PROGRAM S3_01_Motion_43
VAR
	HMI_Motion: FB_HMI_Control;
	Motion: FB_Motion2way;

	tMessageOffset: UINT;
	tNumMessagesPerRow: UINT;
	
	
	MyAdvanceInterlock: BOOL;
	MyReturnInterlock: BOOL;
	
	MyAutoAdvanceCondition: BOOL;
	MyAutoReturnCondition: BOOL;
	testword: WORD;
	myAdvancePrompt: BOOL;
	myReturnPrompt: BOOL;
	advancedSensor: BOOL;
	returnedSensor: BOOL;
	AdvanceCoil: BOOL;
	ReturnCoil: BOOL;
END_VAR

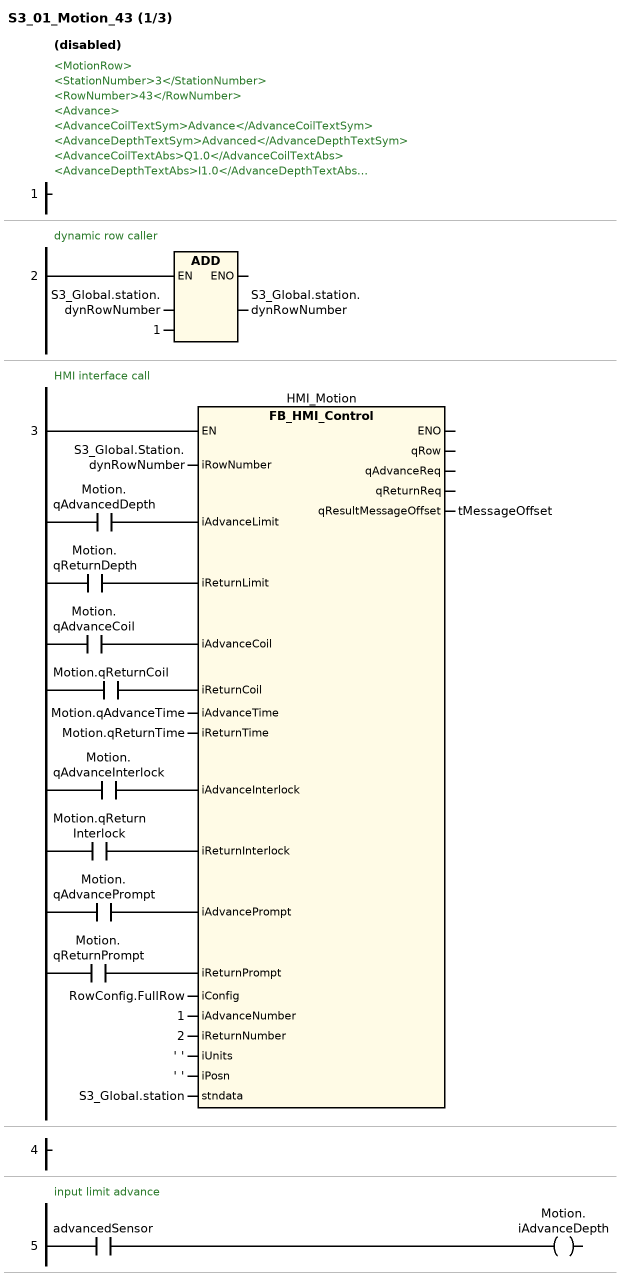
// NETWORK 1 (disabled)
// <MotionRow>
// <StationNumber>3</StationNumber>
// <RowNumber>43</RowNumber>
//   <Advance>
//     <AdvanceCoilTextSym>Advance</AdvanceCoilTextSym>
//     <AdvanceDepthTextSym>Advanced</AdvanceDepthTextSym>
//     <AdvanceCoilTextAbs>Q1.0</AdvanceCoilTextAbs>
//     <AdvanceDepthTextAbs>I1.0</AdvanceDepthTextAbs>
//     <ManSeq>1</ManSeq>
//   </Advance>
//   <Return>
//     <ReturnCoilTextSym>Return</ReturnCoilTextSym>
//     <ReturnDepthTextSym>Returned</ReturnDepthTextSym>
//     <ReturnCoilTextAbs>Q1.1</ReturnCoilTextAbs>
//     <ReturnDepthTextAbs>I1.1</ReturnDepthTextAbs>
//    <ManSeq>2</ManSeq>
//   </Return>
//   <Motion>
//     <NameSym>Clamp Cylinder</NameSym>
//     <NameAbs>A1</NameAbs>
//   </Motion>
// </MotionRow>

// NETWORK 2
// dynamic row caller
S3_Global.station.dynRowNumber := S3_Global.station.dynRowNumber + 1;

// NETWORK 3
// HMI interface call
HMI_Motion(
    iRowNumber := S3_Global.Station.dynRowNumber,
    iAdvanceLimit := Motion.qAdvancedDepth,
    iReturnLimit := Motion.qReturnDepth,
    iAdvanceCoil := Motion.qAdvanceCoil,
    iReturnCoil := Motion.qReturnCoil,
    iAdvanceTime := Motion.qAdvanceTime,
    iReturnTime := Motion.qReturnTime,
    iAdvanceInterlock := Motion.qAdvanceInterlock,
    iReturnInterlock := Motion.qReturnInterlock,
    iAdvancePrompt := Motion.qAdvancePrompt,
    iReturnPrompt := Motion.qReturnPrompt,
    iConfig := RowConfig.FullRow,
    iAdvanceNumber := 1,
    iReturnNumber := 2,
    iUnits := ' ',
    iPosn := ' ',
    stndata := S3_Global.station,
    qResultMessageOffset => tMessageOffset); // FB_HMI_Control

// NETWORK 4

// NETWORK 5
// input limit advance
Motion.iAdvanceDepth := advancedSensor;

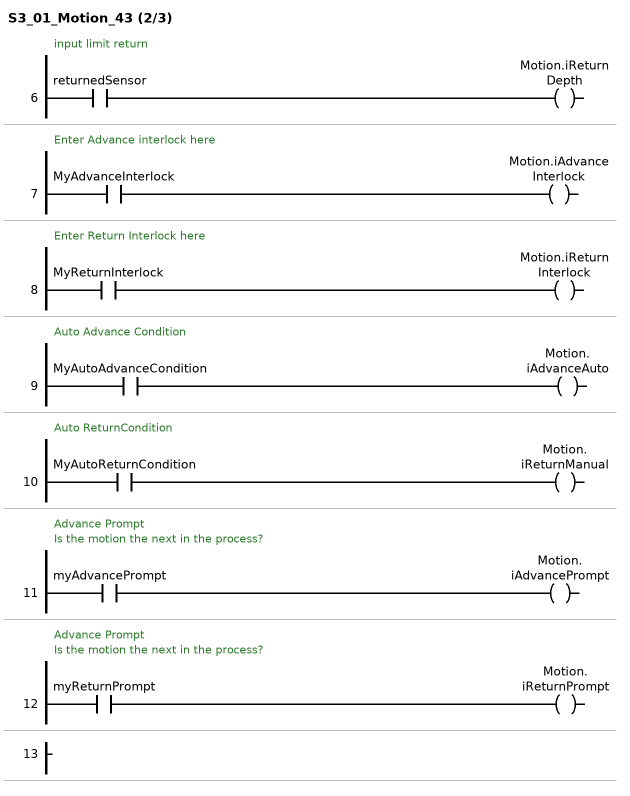
// NETWORK 6
// input limit return
Motion.iReturnDepth := returnedSensor;

// NETWORK 7
// Enter Advance interlock here
Motion.iAdvanceInterlock := MyAdvanceInterlock;

// NETWORK 8
// Enter Return Interlock here
Motion.iReturnInterlock := MyReturnInterlock;

// NETWORK 9
// Auto Advance Condition
Motion.iAdvanceAuto := MyAutoAdvanceCondition;

// NETWORK 10
// Auto ReturnCondition
Motion.iReturnManual := MyAutoReturnCondition;

// NETWORK 11
// Advance Prompt
// Is the motion the next in the process?
Motion.iAdvancePrompt := myAdvancePrompt;

// NETWORK 12
// Advance Prompt
// Is the motion the next in the process?
Motion.iReturnPrompt := myReturnPrompt;

// NETWORK 13

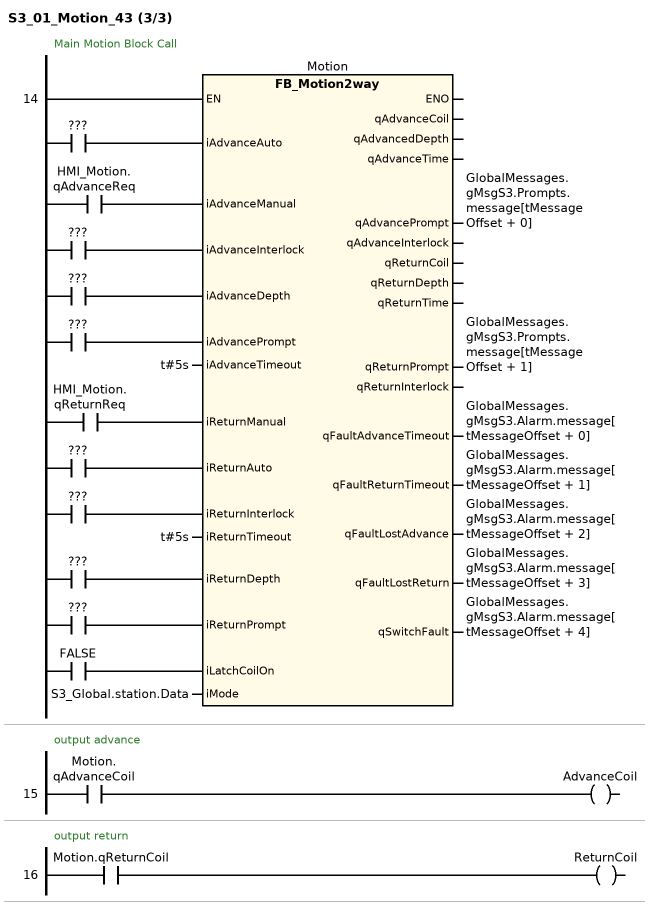
// NETWORK 14
// Main Motion Block Call
Motion(
    iAdvanceManual := HMI_Motion.qAdvanceReq,
    iAdvanceTimeout := t#5s,
    iReturnManual := HMI_Motion.qReturnReq,
    iReturnTimeout := t#5s,
    iLatchCoilOn := FALSE,
    iMode := S3_Global.station.Data,
    qAdvancePrompt => GlobalMessages.gMsgS3.Prompts.message[tMessageOffset + 0],
    qReturnPrompt => GlobalMessages.gMsgS3.Prompts.message[tMessageOffset + 1],
    qFaultAdvanceTimeout => GlobalMessages.gMsgS3.Alarm.message[tMessageOffset + 0],
    qFaultReturnTimeout => GlobalMessages.gMsgS3.Alarm.message[tMessageOffset + 1],
    qFaultLostAdvance => GlobalMessages.gMsgS3.Alarm.message[tMessageOffset + 2],
    qFaultLostReturn => GlobalMessages.gMsgS3.Alarm.message[tMessageOffset + 3],
    qSwitchFault => GlobalMessages.gMsgS3.Alarm.message[tMessageOffset + 4]); // FB_Motion2way

// NETWORK 15
// output advance
AdvanceCoil := Motion.qAdvanceCoil;

// NETWORK 16
// output return
ReturnCoil := Motion.qReturnCoil;

END_PROGRAM

(* stored: Version 1.1.0.1, ProductVersion 3.1.4024.11
   POU S3_01_Motion_43: Id {25c0e845-0274-0390-105c-e67ff9951cfc}, SpecialFunc None *)
